TEXTLIST Recipt_no
  1 = 'Recipe 1'
  2 = 'Recipe 2'
  3 = 'Recipe 3'
  4 = 'Recipe 4'
  5 = 'Recipe 5'
  6 = 'Recipe 6'
  7 = 'Recipe 7'
  8 = 'Recipe 8'
  9 = 'Recipe 9'
  10 = 'Recipe 10'
   = ''
END_TEXTLIST

(* stored: Version 1.1.0.1, ProductVersion 3.1.4024.11
   TextList Recipt_no: Id {c9a7465f-028d-4405-b3b2-b5a7440b2331} *)
